RoboDK station: Sheet A on table.rdk

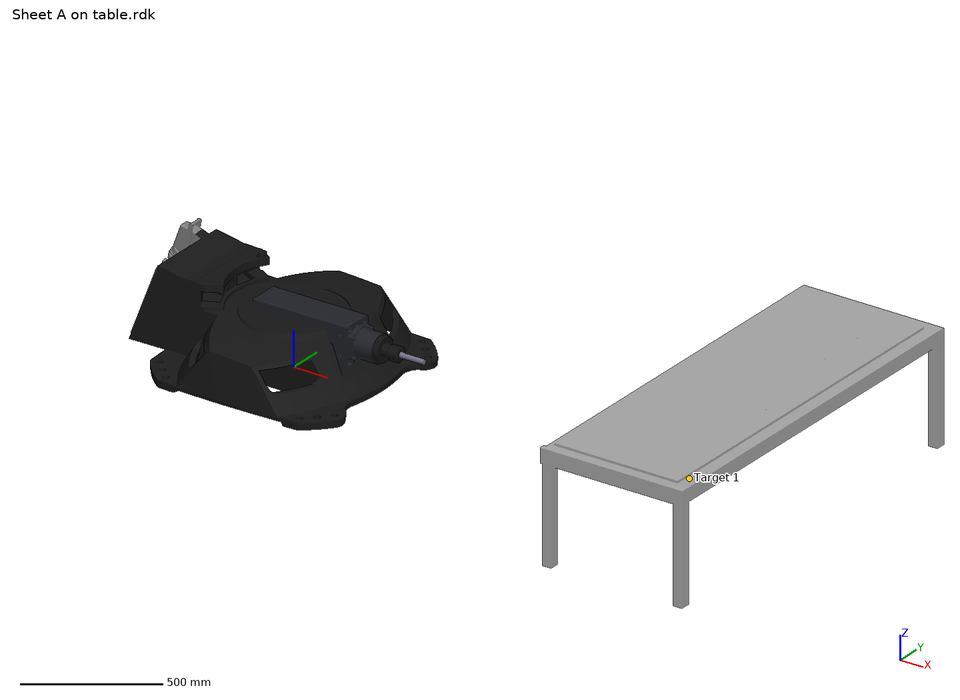
[picture v0: the station drawn from its stored meshes, robots at their saved joint values, targets as dots, program paths as lines]
Station Sheet A on table (saved by RoboDK 5.2.3). Poses are relative to the parent item; angles as X-Y-Z fixed-axis rotations.
  - frame KUKA KR 210 R2700 extra Base at (0, 0, 0) mm
    - robot KUKA KR 210 R2700 extra: 6 axes, payload 210 kg, reach 2696 mm, repeatability 0.06 mm, weight 1068 kg
        joint limits [-185, -140, -120, -350, -125, -350] to [185, -5, 155, 350, 125, 350]; home [0, -90, 90, 0, 0, 0]; saved at [0, -90, 90, 0, 0, 0]
      - tool Spindle, TCP at (557.2, 0, 176) mm, rotated rx 0 ry 90 rz 0 deg, size 692.9 x 170 x 256 mm
    - target Target 1 (Cartesian target) at (2182, -700, 455.5) mm, rotated rx -180 ry 0 rz 180 deg; joints [21.348, -60.261, 91.697, 36.848, -37.375, -30.775] of KUKA KR 210 R2700 extra
  - object Table at (1640, -780, 0) mm, size 610 x 1605 x 465 mm
  - object sheet A at (2172.9, 5, 455) mm, rotated rx 0 ry 0 rz 90 deg, size 1500 x 148.4 x 0.8 mm, geometry from sheet A.stl
